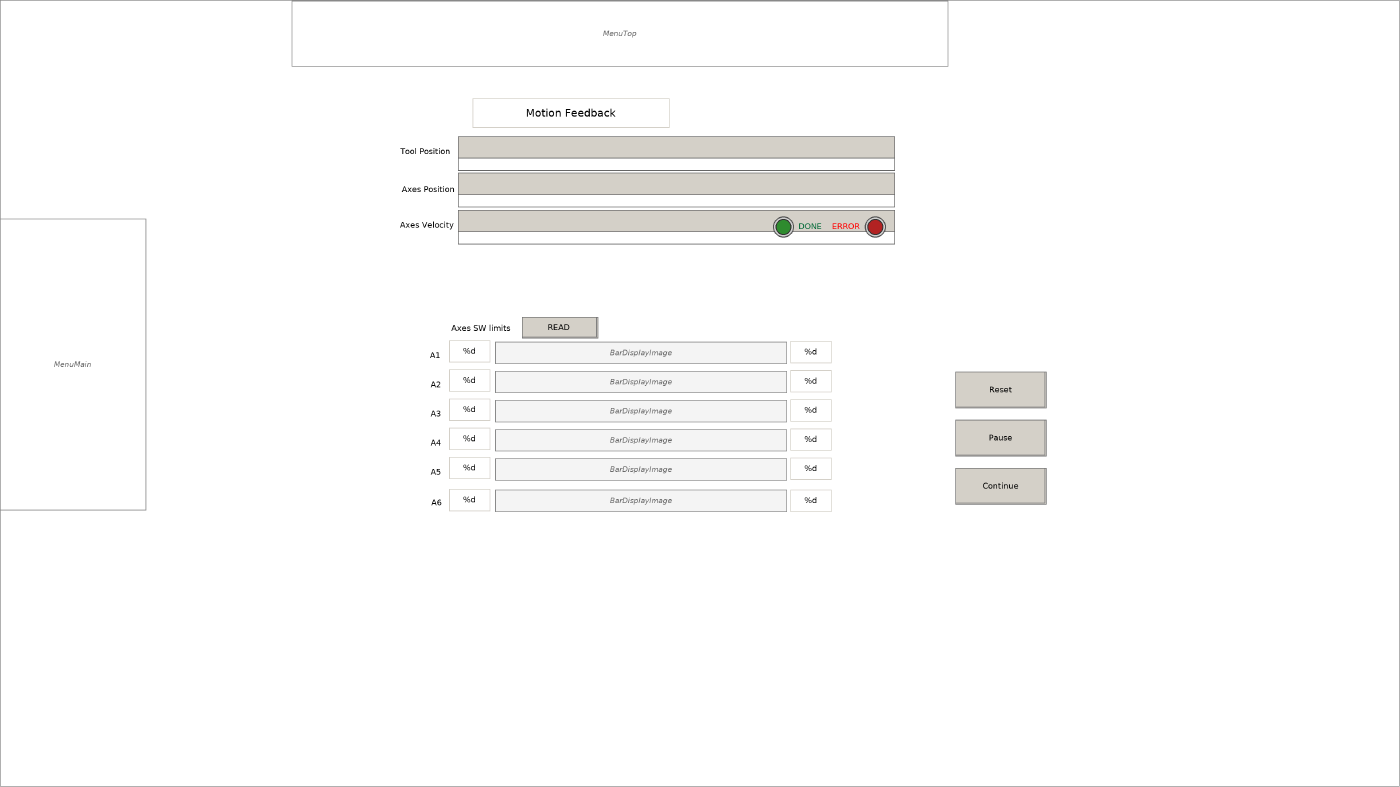
VISUALIZATION Motion_FBK  // 1920x1080
    Frame (400,1 900x90)
        shows MenuTop()
    Frame (0,300 200x400)
        shows MenuMain()
    Textfield (648,135 270x40), "Motion Feedback"
    Table (628,237 599x47), data array: GVL.HMI_ActualAxisPosition
        p3854506369: GVL.HMI_ActualAxisPosition.A1
        p1892666644: GVL.HMI_ActualAxisPosition.A2
        p338671338: GVL.HMI_ActualAxisPosition.A3
        p2170511999: GVL.HMI_ActualAxisPosition.A4
        p3723444502: GVL.HMI_ActualAxisPosition.A5
        p1218418051: GVL.HMI_ActualAxisPosition.A6
        p746581629: GVL.HMI_ActualAxisPosition.E1
        p3104783080: GVL.HMI_ActualAxisPosition.E2
        p2501879983: GVL.HMI_ActualAxisPosition.E3
        p7306298: GVL.HMI_ActualAxisPosition.E4
        p1933151965: GVL.HMI_ActualAxisPosition.E5
        p3863566920: GVL.HMI_ActualAxisPosition.E6
        p2192122294: ActualKarthPositon.E5
        p400160035: ActualKarthPositon.E6
    Table (628,187 599x47), data array: mxA_Motion.fbKRC_ReadActualPosition.Position
        p3854506369: mxA_Motion.fbKRC_ReadActualPosition.Position.X
        p1892666644: mxA_Motion.fbKRC_ReadActualPosition.Position.Y
        p338671338: mxA_Motion.fbKRC_ReadActualPosition.Position.Z
        p2170511999: mxA_Motion.fbKRC_ReadActualPosition.Position.A
        p3723444502: mxA_Motion.fbKRC_ReadActualPosition.Position.B
        p1218418051: mxA_Motion.fbKRC_ReadActualPosition.Position.C
        p746581629: mxA_Motion.fbKRC_ReadActualPosition.Position.Status
        p3104783080: mxA_Motion.fbKRC_ReadActualPosition.Position.Turn
        p2501879983: mxA_Motion.fbKRC_ReadActualPosition.Position.E1
        p7306298: mxA_Motion.fbKRC_ReadActualPosition.Position.E2
        p1933151965: mxA_Motion.fbKRC_ReadActualPosition.Position.E3
        p3863566920: mxA_Motion.fbKRC_ReadActualPosition.Position.E4
        p2192122294: mxA_Motion.fbKRC_ReadActualPosition.Position.E5
        p400160035: mxA_Motion.fbKRC_ReadActualPosition.Position.E6
        p4092479075: Rx
        p2237128397: Ry
        p505689113: Rz
        p1757482276: status
        p4088588272: turn
    Rectangle (537,193 93x30), "Tool Position"
    Rectangle (541,245 93x30), "Axes Position"
    BarDisplayImage (679,469 400x30), value: mxA_Motion.fbKRC_ReadActualAxisPosition.A1, style: BarDisplayImage-Gray, scale format: %.1f, scale -180..180
    BarDisplayImage (679,509 400x30), value: mxA_Motion.fbKRC_ReadActualAxisPosition.A2, style: BarDisplayImage-Gray, scale format: %.1f, scale -180..180
    BarDisplayImage (679,549 400x30), value: mxA_Motion.fbKRC_ReadActualAxisPosition.A3, style: BarDisplayImage-Gray, scale format: %.1f, scale -180..180
    BarDisplayImage (679,589 400x30), value: mxA_Motion.fbKRC_ReadActualAxisPosition.A4, style: BarDisplayImage-Gray, scale format: %.1f, scale -360..360
    BarDisplayImage (679,629 400x30), value: mxA_Motion.fbKRC_ReadActualAxisPosition.A5, style: BarDisplayImage-Gray, scale format: %.1f, scale -180..180
    BarDisplayImage (679,672 400x30), value: mxA_Motion.fbKRC_ReadActualAxisPosition.A6, style: BarDisplayImage-Gray, scale format: %.1f, scale -360..360
    Label (580,476 34x24), "A1"
    Label (581,516 34x24), "A2"
    Label (581,556 34x24), "A3"
    Label (581,596 34x24), "A4"
    Label (581,636 34x24), "A5"
    Label (582,678 34x24), "A6"
    Rectangle (603,430 113x41), "Axes SW limits"
    Textfield (1084,468 56x30), "%d", text variable: MAIN.Read_Axes_SW_Limts.A1_Max
    Textfield (1084,508 56x30), "%d", text variable: MAIN.Read_Axes_SW_Limts.A2_Max
    Textfield (1084,548 56x30), "%d", text variable: MAIN.Read_Axes_SW_Limts.A3_Max
    Textfield (1084,588 56x30), "%d", text variable: MAIN.Read_Axes_SW_Limts.A4_Max
    Textfield (1084,628 56x30), "%d", text variable: MAIN.Read_Axes_SW_Limts.A5_Max
    Textfield (1084,672 56x30), "%d", text variable: MAIN.Read_Axes_SW_Limts.A6_Max
    Textfield (616,467 56x30), "%d", text variable: MAIN.Read_Axes_SW_Limts.A1_Min
    Textfield (616,507 56x30), "%d", text variable: MAIN.Read_Axes_SW_Limts.A2_Min
    Textfield (616,547 56x30), "%d", text variable: MAIN.Read_Axes_SW_Limts.A3_Min
    Textfield (616,587 56x30), "%d", text variable: MAIN.Read_Axes_SW_Limts.A4_Min
    Textfield (616,627 56x30), "%d", text variable: MAIN.Read_Axes_SW_Limts.A5_Min
    Textfield (616,671 56x30), "%d", text variable: MAIN.Read_Axes_SW_Limts.A6_Min
    Button (716,435 104x29), "READ"
        OnMouseClick: toggle MAIN.Read_Axes_SW_Limts.ExecuteCmd
    Button (1310,576 125x50), "Pause"
        tap mxA_Motion.fbAutoDemo.fbKRC_Interrupt.Execute
    Button (1310,642 125x50), "Continue"
        tap mxA_Motion.fbAutoDemo.fbKRC_Continue.Enable
    Button (1310,510 125x50), "Reset"
        tap MAIN.Write_Program_Abort.ExecuteCmd
    Table (628,288 599x47), data array: Read_Axes_Velocity.ReadAxesVelocity
        p3854506369: Read_Axes_Velocity.ReadAxesVelocity.AxisGroupIdx
        p1892666644: Read_Axes_Velocity.ReadAxesVelocity.ExecuteCmd
        p338671338: Read_Axes_Velocity.ReadAxesVelocity.Done
        p2170511999: Read_Axes_Velocity.ReadAxesVelocity.Error
        p3723444502: Read_Axes_Velocity.ReadAxesVelocity.ErrorID
        p1218418051: Read_Axes_Velocity.ReadAxesVelocity.A1
        p746581629: Read_Axes_Velocity.ReadAxesVelocity.A2
        p3104783080: Read_Axes_Velocity.ReadAxesVelocity.A3
        p2501879983: Read_Axes_Velocity.ReadAxesVelocity.A4
        p7306298: Read_Axes_Velocity.ReadAxesVelocity.A5
        p1933151965: Read_Axes_Velocity.ReadAxesVelocity.A6
        p3863566920: Read_Axes_Velocity.ReadAxesVelocity.E1
        p2192122294: Read_Axes_Velocity.ReadAxesVelocity.E2
        p400160035: Read_Axes_Velocity.ReadAxesVelocity.E3
        p1265227338: Read_Axes_Velocity.ReadAxesVelocity.E4
        p3726181087: Read_Axes_Velocity.ReadAxesVelocity.E5
        p3136911649: Read_Axes_Velocity.ReadAxesVelocity.E6
        p797552052: Read_Axes_Velocity.ReadAxesVelocity.mxA_ExecuteCommand
    Rectangle (539,294 93x30), "Axes Velocity"
    Lamp1 (1058,295 33x33), variable: Read_Axes_Velocity.ReadAxesVelocity.Done, style: Lamp-Lamp1-Green
    Lamp1 (1184,295 33x33), variable: Read_Axes_Velocity.ReadAxesVelocity.Error, style: Lamp-Lamp1-Red
    Rectangle (1088,300 46x22), "DONE"
    Rectangle (1137,300 46x22), "ERROR"
END_VISUALIZATION

(* stored: Version 1.1.0.1, ProductVersion 3.1.4024.10
   Visu Motion_FBK: Id {77dfa8c5-424c-4d55-a891-efd15dba6c6c} *)
